(* Logix 5000 project; controller full_alarm_and_fault_management_system vendor 1 type 14 code 196 rev 36.11; software revision 36.00 *)

TASK MainTask (continuous, watchdog 500 ms) : MainProgram

MODULES
   Local : vendor 1 type 14 code 196 (5069 0, rev 36.11)
END_MODULES

PROGRAM MainProgram   (* main routine MainRoutine *)
VAR
   Active_Temp_SP : DINT;
   Code_EStop : DINT;   // 1001
   Code_HighLevel : DINT;   // 1005
   Code_HighTemp : DINT;   // 1003
   Code_LowLevel : DINT;   // 1006
   Code_LowTemp : DINT;   // 1004
   Code_MotorOL : DINT;   // 1002
   Code_SensorFault : DINT;   // 1010
   Code_Valve1Fail : DINT;   // 1007
   Code_Valve2Fail : DINT;   // 1008
   Code_Valve3Fail : DINT;   // 1009
   Current_Fault_Code : DINT;   // Optional displayed fault code
   Fault_Count : DINT;   // Optional number of active faults
   Flow_1_ok : BOOL;
   Flow_2_Ok : BOOL;
   Flow_3_ok : BOOL;
   Heat_Enable : BOOL;
   machine_Runpermissive : BOOL;
   ONS_EStop_TS : BOOL;   // One-shot storage for E-stop tiimestamping
   ONS_HighLevel_TS : BOOL;   // One-shot storage for high level timestamp
   ONS_HighTemp_TS : BOOL;   // One-shot storage for High temp timestamp
   ONS_LowLevel_TS : BOOL;   // One-shot storage for low level timestamp
   ONS_LowTemp_TS : BOOL;   // One-shot storage for low temp timestamp
   ONS_MotorOL_TS : BOOL;   // One-shot storage for motor overload timestamp
   ONS_Reset : BOOL;   // One-shot storage for reset pushbutton
   ONS_Sensor_TS : BOOL;   // One-shot storage for sensor fault timestamp
   ONS_Valve1_TS : BOOL;   // One-shot storage for valve 1 fault timestamp
   ONS_Valve2_TS : BOOL;   // One-shot storage for valve 2 fault timestamp
   ONS_Valve3_TS : BOOL;   // One-shot storage for valve 3 fault timestamp
   Sim_EStop_PB : BOOL;
   Sim_MotorOL : BOOL;
   system_run : BOOL;
   T_HeatTimeout : TIMER;
   Temp_PV : DINT;
   valve_1 : BOOL;
   valve_2 : BOOL;
   valve_3 : BOOL;
END_VAR
VAR_OUTPUT
   AlarmHorn : BOOL;   // Alarm output
   Any_Fault_Active : BOOL;   // True if any fault is latched
   Fault_Reset_Request : BOOL;   // One-shot reset request
   Flt_EStop : BOOL;   // Latched E-stop fault
   Flt_HighLevel : BOOL;   // Latched high level fault
   Flt_HighTemp : BOOL;   // Latched high temp fault
   Flt_LowLevel : BOOL;   // Latched low level fault
   Flt_LowTemp : BOOL;   // Latched low temp fault
   Flt_MotorOL : BOOL;   // Latched motor overload fault
   Flt_SensorFault : BOOL;   // Latched sensor fault
   Flt_Valve1Fail : BOOL;   // Latched valve 1 failure
   Flt_Valve2Fail : BOOL;   // latched valve 2 failure
   Flt_Valve3Fail : BOOL;   // Latched valve 3 failure
   Rst_OKLowLevel : BOOL;   // Low level cleared
   RstOk_EStop : BOOL;   // E-stop cleared, reset allowed
   RstOK_HighLevel : BOOL;   // High level cleared
   RstOK_HighTemp : BOOL;   // High temp cleared
   RstOK_LowTemp : BOOL;   // Low Temp cleared
   RstOk_motorOL : BOOL;   // Motor overload cleared
   RstOK_SensorFault : BOOL;   // sensor fault cleared
   RstOK_Valve1Fail : BOOL;   // Valve 1 fault cleared
   RstOK_Valve2Fail : BOOL;   // Valve 2 fault cleared
   RstOK_Valve3Fail : BOOL;   // Valve 3 fault cleared
   RTC_DateTime : DINT[7];   // Current controller time component
   TS_EStop : DINT[7];   // Timestamp for e-stop fault
   TS_HighLevel : DINT[7];   // Timestamp for high level
   TS_HighTemp : DINT[7];   // Timestamp for high temp
   TS_LowLevel : DINT[7];   // Timestamp for low level
   TS_LowTemp : DINT[7];   // Timestamp for low temp
   TS_MotorOL : DINT[7];   // Timestamp for motor overload
   TS_SensorFault : DINT[7];   // Timestamp for sensor fault
   TS_Valve1Fail : DINT[7];   // Timestamp for valve 1 fault
   TS_Valve2Fail : DINT[7];   // Timestamp for valve 2 Fault
   TS_Valve3Fail : DINT[7];   // Timestamp for valve 3 fault
END_VAR
VAR_INPUT
   Cond_EStop : BOOL;   // Raw E-stop condition
   Cond_Highlevel : BOOL;   // Raw high level fault
   Cond_HighTemp : BOOL;   // Raw high temperature fault
   Cond_Lowlevel : BOOL;   // Raw low level fault
   Cond_LowTemp : BOOL;   // Raw low temp fault
   Cond_MotorOL : BOOL;   // Raw motor overload condition
   Cond_SensorFault : BOOL;   // Raw valve 3 failure
   Cond_Valve1Fail : BOOL;   // Raw low level fault
   Cond_Valve2Fail : BOOL;   // Raw valve 1 failure
   Cond_Valve3Fail : BOOL;   // Raw valve 2 failure
   PB_AckFaults : BOOL;   // Optional acknowledge pushbutton
   PB_ResetFaults : BOOL;   // operator fault reset pushbutton
   Tank_level : DINT;
END_VAR

ROUTINE Fault_Detection   (* ladder *)
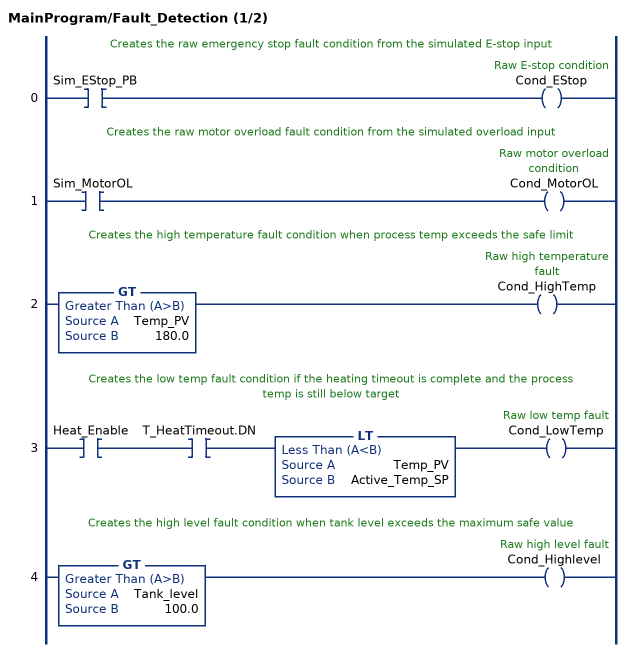
   // Creates the raw emergency stop fault condition from the simulated E-stop input
   0: XIC(Sim_EStop_PB)OTE(Cond_EStop);
   // Creates the raw motor overload fault condition from the simulated overload input
   1: XIC(Sim_MotorOL)OTE(Cond_MotorOL);
   // Creates the high temperature fault condition when process temp exceeds the safe limit
   2: GT(Temp_PV,180.0)OTE(Cond_HighTemp);
   // Creates the low temp fault condition if the heating timeout is complete and the process temp is still below target
   3: XIC(Heat_Enable)XIC(T_HeatTimeout.DN)LT(Temp_PV,Active_Temp_SP)OTE(Cond_LowTemp);
   // Creates the high level fault condition when tank level exceeds the maximum safe value
   4: GT(Tank_level,100.0)OTE(Cond_Highlevel);
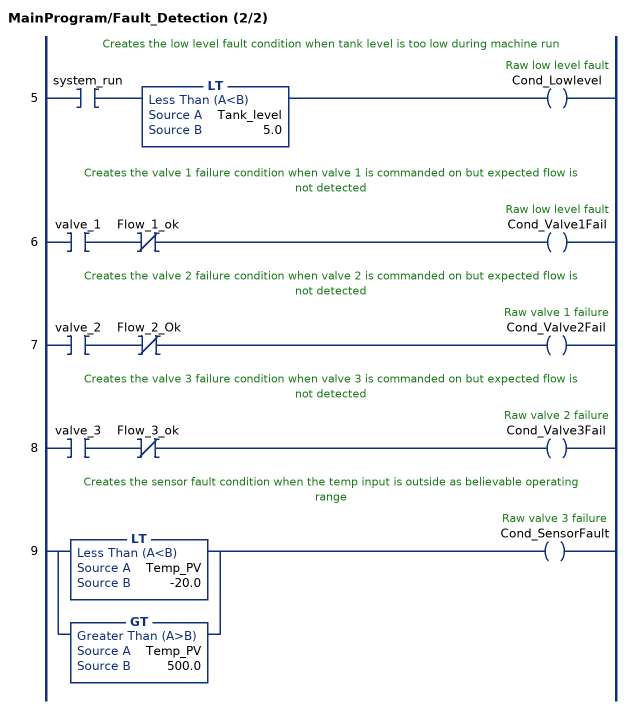
   // Creates the low level fault condition when tank level is too low during machine run
   5: XIC(system_run)LT(Tank_level,5.0)OTE(Cond_Lowlevel);
   // Creates the valve 1 failure condition when valve 1 is commanded on but expected flow is not detected
   6: XIC(valve_1)XIO(Flow_1_ok)OTE(Cond_Valve1Fail);
   // Creates the valve 2 failure condition when valve 2 is commanded on but expected flow is not detected
   7: XIC(valve_2)XIO(Flow_2_Ok)OTE(Cond_Valve2Fail);
   // Creates the valve 3 failure condition when valve 3 is commanded on but expected flow is not detected
   8: XIC(valve_3)XIO(Flow_3_ok)OTE(Cond_Valve3Fail);
   // Creates the sensor fault condition when the temp input is outside as believable operating range
   9: [LT(Temp_PV,-20.0) ,GT(Temp_PV,500.0) ]OTE(Cond_SensorFault);
END_ROUTINE

ROUTINE Fault_Display   (* ladder *)
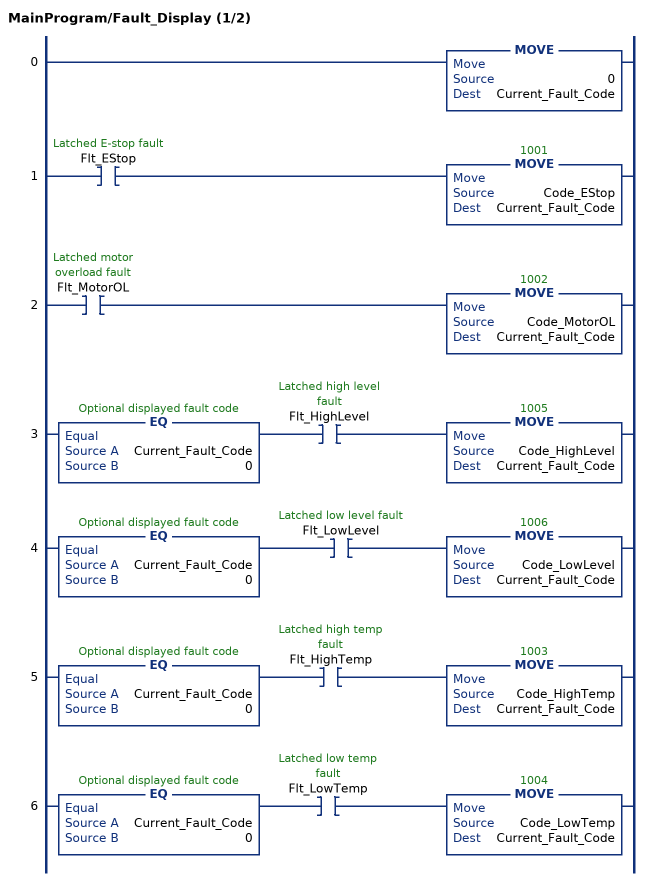
   0: MOVE(0,Current_Fault_Code);
   1: XIC(Flt_EStop)MOVE(Code_EStop,Current_Fault_Code);
   2: XIC(Flt_MotorOL)MOVE(Code_MotorOL,Current_Fault_Code);
   3: EQ(Current_Fault_Code,0)XIC(Flt_HighLevel)MOVE(Code_HighLevel,Current_Fault_Code);
   4: EQ(Current_Fault_Code,0)XIC(Flt_LowLevel)MOVE(Code_LowLevel,Current_Fault_Code);
   5: EQ(Current_Fault_Code,0)XIC(Flt_HighTemp)MOVE(Code_HighTemp,Current_Fault_Code);
   6: EQ(Current_Fault_Code,0)XIC(Flt_LowTemp)MOVE(Code_LowTemp,Current_Fault_Code);
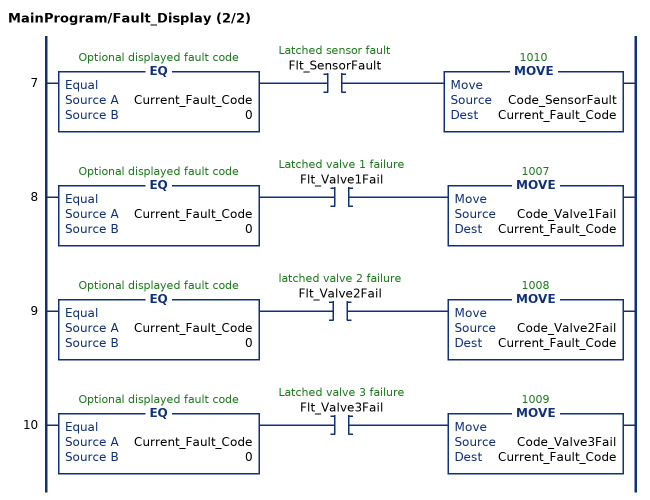
   7: EQ(Current_Fault_Code,0)XIC(Flt_SensorFault)MOVE(Code_SensorFault,Current_Fault_Code);
   8: EQ(Current_Fault_Code,0)XIC(Flt_Valve1Fail)MOVE(Code_Valve1Fail,Current_Fault_Code);
   9: EQ(Current_Fault_Code,0)XIC(Flt_Valve2Fail)MOVE(Code_Valve2Fail,Current_Fault_Code);
   10: EQ(Current_Fault_Code,0)XIC(Flt_Valve3Fail)MOVE(Code_Valve3Fail,Current_Fault_Code);
END_ROUTINE

ROUTINE Fault_Latching   (* ladder *)
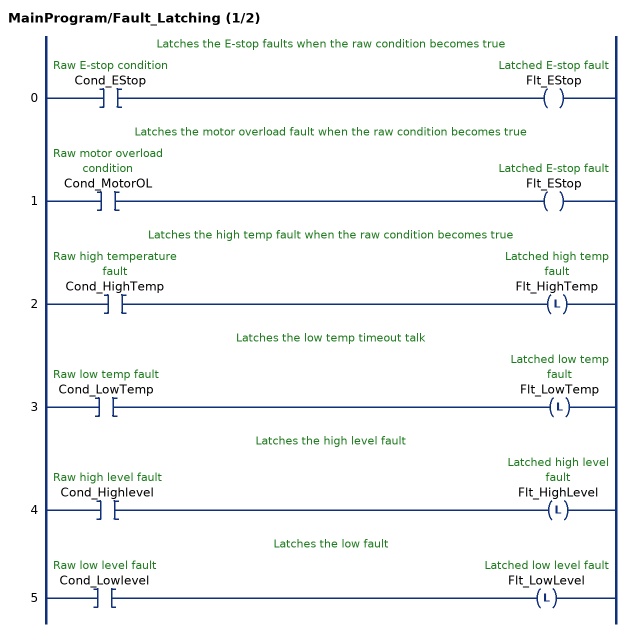
   // Latches the E-stop faults when the raw condition becomes true
   0: XIC(Cond_EStop)OTE(Flt_EStop);
   // Latches the motor overload fault when the raw condition becomes true
   1: XIC(Cond_MotorOL)OTE(Flt_EStop);
   // Latches the high temp fault when the raw condition becomes true
   2: XIC(Cond_HighTemp)OTL(Flt_HighTemp);
   // Latches the low temp timeout talk
   3: XIC(Cond_LowTemp)OTL(Flt_LowTemp);
   // Latches the high level fault
   4: XIC(Cond_Highlevel)OTL(Flt_HighLevel);
   // Latches the low fault
   5: XIC(Cond_Lowlevel)OTL(Flt_LowLevel);
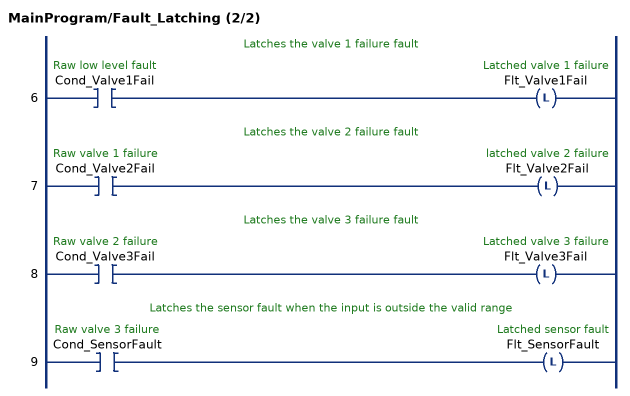
   // Latches the valve 1 failure fault
   6: XIC(Cond_Valve1Fail)OTL(Flt_Valve1Fail);
   // Latches the valve 2 failure fault
   7: XIC(Cond_Valve2Fail)OTL(Flt_Valve2Fail);
   // Latches the valve 3 failure fault
   8: XIC(Cond_Valve3Fail)OTL(Flt_Valve3Fail);
   // Latches the sensor fault when the input is outside the valid range
   9: XIC(Cond_SensorFault)OTL(Flt_SensorFault);
END_ROUTINE

ROUTINE Fault_Reset   (* ladder *)
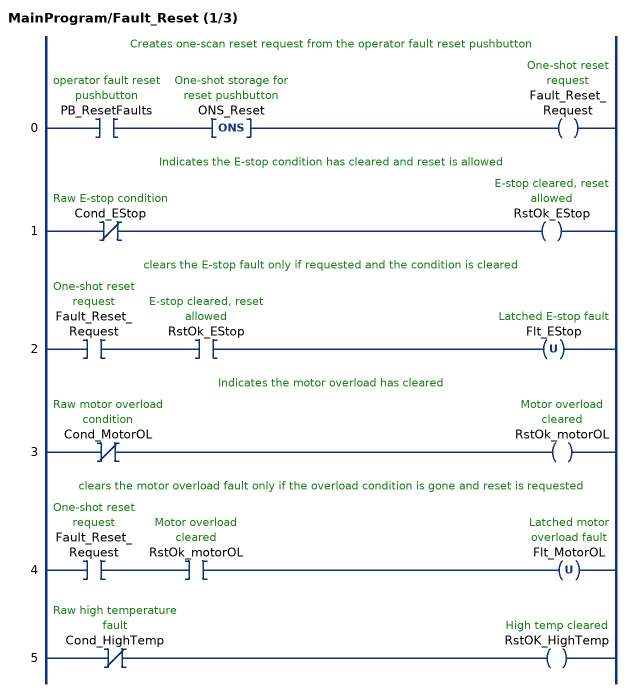
   // Creates one-scan reset request from the operator fault reset pushbutton
   0: XIC(PB_ResetFaults)ONS(ONS_Reset)OTE(Fault_Reset_Request);
   // Indicates the E-stop condition has cleared and reset is allowed
   1: XIO(Cond_EStop)OTE(RstOk_EStop);
   // clears the E-stop fault only if requested and the condition is cleared
   2: XIC(Fault_Reset_Request)XIC(RstOk_EStop)OTU(Flt_EStop);
   // Indicates the motor overload has cleared
   3: XIO(Cond_MotorOL)OTE(RstOk_motorOL);
   // clears the motor overload fault only if the overload condition is gone and reset is requested
   4: XIC(Fault_Reset_Request)XIC(RstOk_motorOL)OTU(Flt_MotorOL);
   5: XIO(Cond_HighTemp)OTE(RstOK_HighTemp);
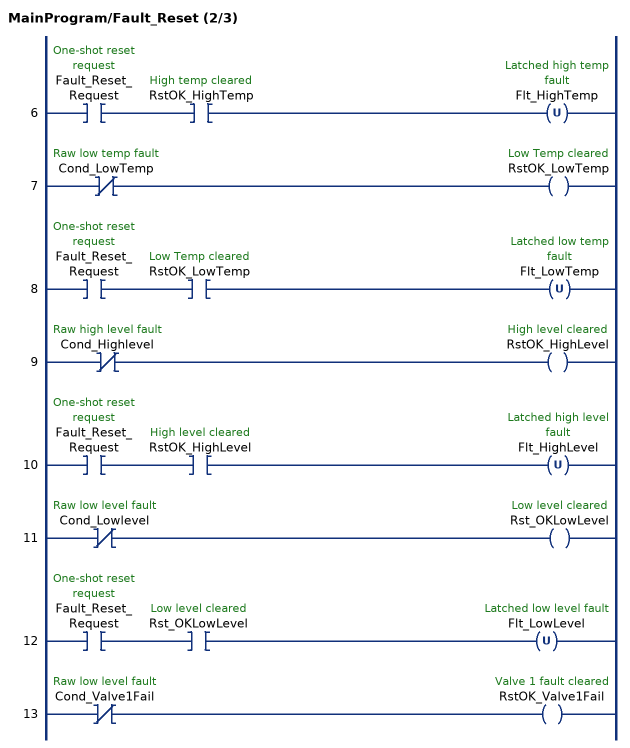
   6: XIC(Fault_Reset_Request)XIC(RstOK_HighTemp)OTU(Flt_HighTemp);
   7: XIO(Cond_LowTemp)OTE(RstOK_LowTemp);
   8: XIC(Fault_Reset_Request)XIC(RstOK_LowTemp)OTU(Flt_LowTemp);
   9: XIO(Cond_Highlevel)OTE(RstOK_HighLevel);
   10: XIC(Fault_Reset_Request)XIC(RstOK_HighLevel)OTU(Flt_HighLevel);
   11: XIO(Cond_Lowlevel)OTE(Rst_OKLowLevel);
   12: XIC(Fault_Reset_Request)XIC(Rst_OKLowLevel)OTU(Flt_LowLevel);
   13: XIO(Cond_Valve1Fail)OTE(RstOK_Valve1Fail);
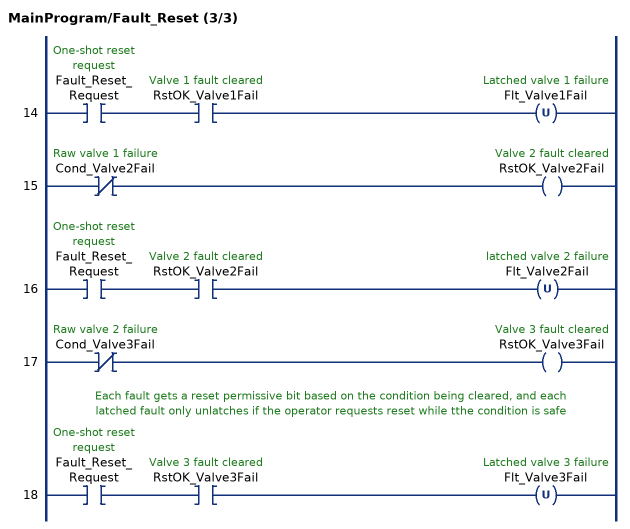
   14: XIC(Fault_Reset_Request)XIC(RstOK_Valve1Fail)OTU(Flt_Valve1Fail);
   15: XIO(Cond_Valve2Fail)OTE(RstOK_Valve2Fail);
   16: XIC(Fault_Reset_Request)XIC(RstOK_Valve2Fail)OTU(Flt_Valve2Fail);
   17: XIO(Cond_Valve3Fail)OTE(RstOK_Valve3Fail);
   // Each fault gets a reset permissive bit based on the condition being cleared, and each latched fault only unlatches if the operator requests reset while tthe condition is safe
   18: XIC(Fault_Reset_Request)XIC(RstOK_Valve3Fail)OTU(Flt_Valve3Fail);
END_ROUTINE

ROUTINE Fault_summary   (* ladder *)
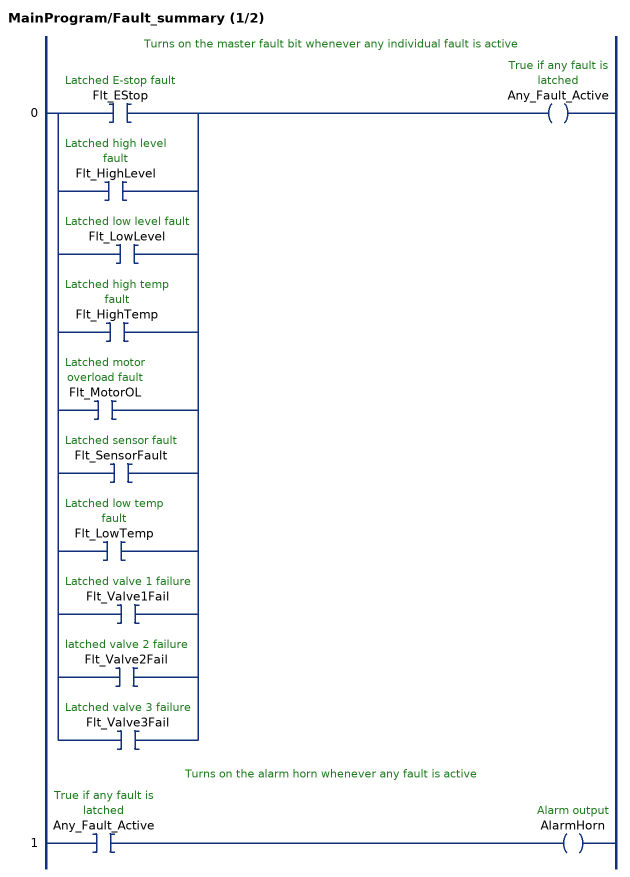
   // Turns on the master fault bit whenever any individual fault is active
   0: [XIC(Flt_EStop) ,XIC(Flt_HighLevel) ,XIC(Flt_LowLevel) ,XIC(Flt_HighTemp) ,XIC(Flt_MotorOL) ,XIC(Flt_SensorFault) ,XIC(Flt_LowTemp) ,XIC(Flt_Valve1Fail) ,XIC(Flt_Valve2Fail) ,XIC(Flt_Valve3Fail) ]OTE(Any_Fault_Active);
   // Turns on the alarm horn whenever any fault is active
   1: XIC(Any_Fault_Active)OTE(AlarmHorn);
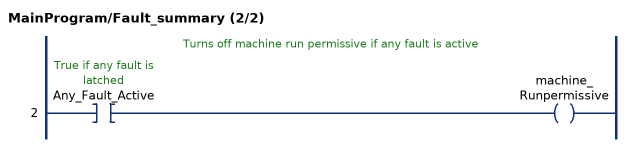
   // Turns off machine run permissive if any fault is active
   2: XIC(Any_Fault_Active)OTE(machine_Runpermissive);
END_ROUTINE

ROUTINE Fault_Timestamps   (* ladder *)
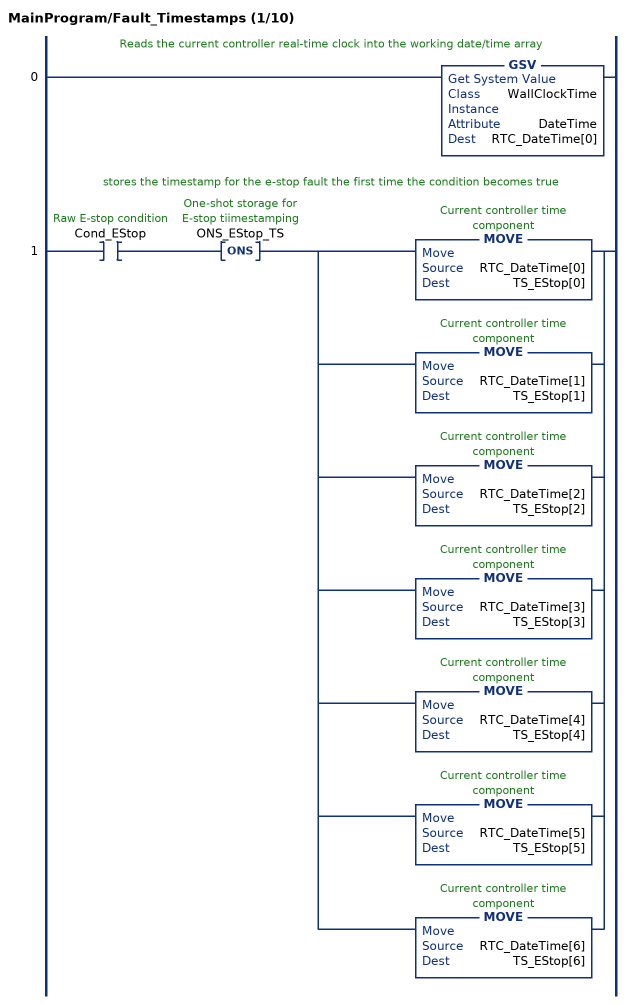
   // Reads the current controller real-time clock into the working date/time array
   0: GSV(WallClockTime,,DateTime,RTC_DateTime[0]);
   // stores the timestamp for the e-stop fault the first time the condition becomes true
   1: XIC(Cond_EStop)ONS(ONS_EStop_TS)[MOVE(RTC_DateTime[0],TS_EStop[0]) ,MOVE(RTC_DateTime[1],TS_EStop[1]) ,MOVE(RTC_DateTime[2],TS_EStop[2]) ,MOVE(RTC_DateTime[3],TS_EStop[3]) ,MOVE(RTC_DateTime[4],TS_EStop[4]) ,MOVE(RTC_DateTime[5],TS_EStop[5]) ,MOVE(RTC_DateTime[6],TS_EStop[6]) ];
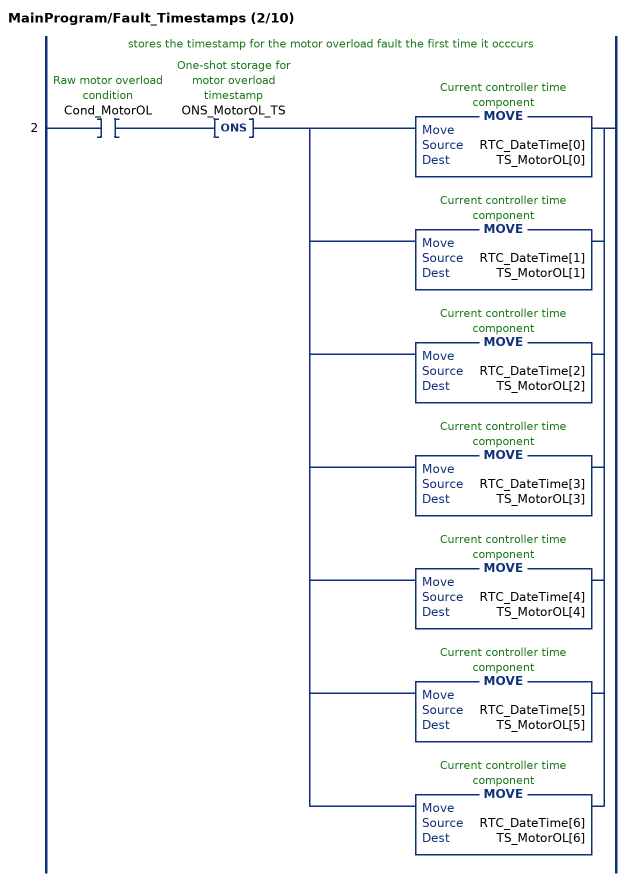
   // stores the timestamp for the motor overload fault the first time it occcurs
   2: XIC(Cond_MotorOL)ONS(ONS_MotorOL_TS)[MOVE(RTC_DateTime[0],TS_MotorOL[0]) ,MOVE(RTC_DateTime[1],TS_MotorOL[1]) ,MOVE(RTC_DateTime[2],TS_MotorOL[2]) ,MOVE(RTC_DateTime[3],TS_MotorOL[3]) ,MOVE(RTC_DateTime[4],TS_MotorOL[4]) ,MOVE(RTC_DateTime[5],TS_MotorOL[5]) ,MOVE(RTC_DateTime[6],TS_MotorOL[6]) ];
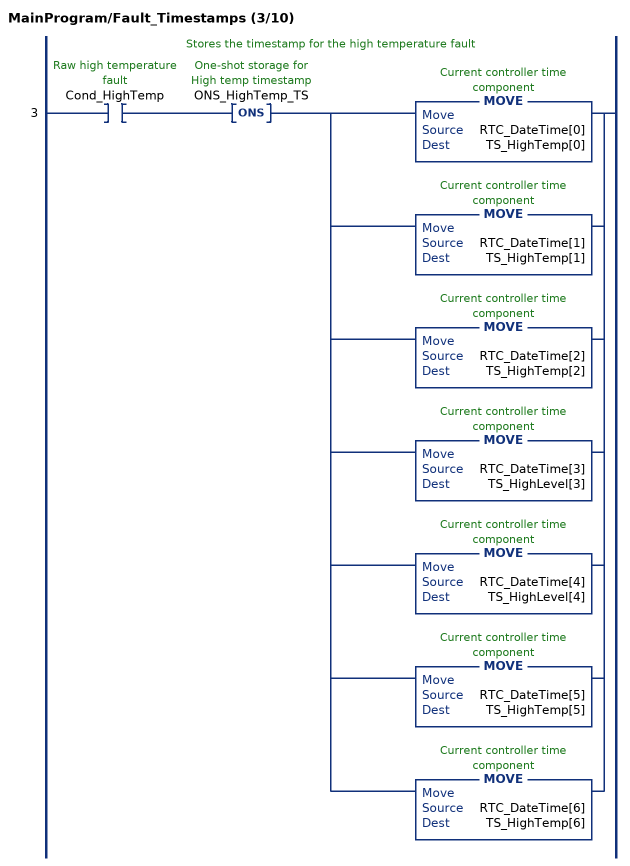
   // Stores the timestamp for the high temperature fault
   3: XIC(Cond_HighTemp)ONS(ONS_HighTemp_TS)[MOVE(RTC_DateTime[0],TS_HighTemp[0]) ,MOVE(RTC_DateTime[1],TS_HighTemp[1]) ,MOVE(RTC_DateTime[2],TS_HighTemp[2]) ,MOVE(RTC_DateTime[3],TS_HighLevel[3]) ,MOVE(RTC_DateTime[4],TS_HighLevel[4]) ,MOVE(RTC_DateTime[5],TS_HighTemp[5]) ,MOVE(RTC_DateTime[6],TS_HighTemp[6]) ];
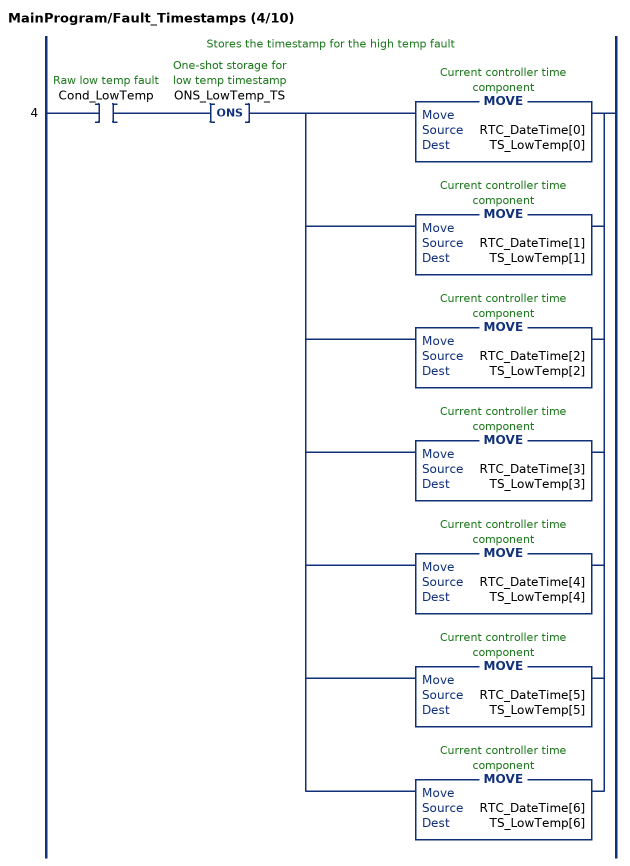
   // Stores the timestamp for the high temp fault
   4: XIC(Cond_LowTemp)ONS(ONS_LowTemp_TS)[MOVE(RTC_DateTime[0],TS_LowTemp[0]) ,MOVE(RTC_DateTime[1],TS_LowTemp[1]) ,MOVE(RTC_DateTime[2],TS_LowTemp[2]) ,MOVE(RTC_DateTime[3],TS_LowTemp[3]) ,MOVE(RTC_DateTime[4],TS_LowTemp[4]) ,MOVE(RTC_DateTime[5],TS_LowTemp[5]) ,MOVE(RTC_DateTime[6],TS_LowTemp[6]) ];
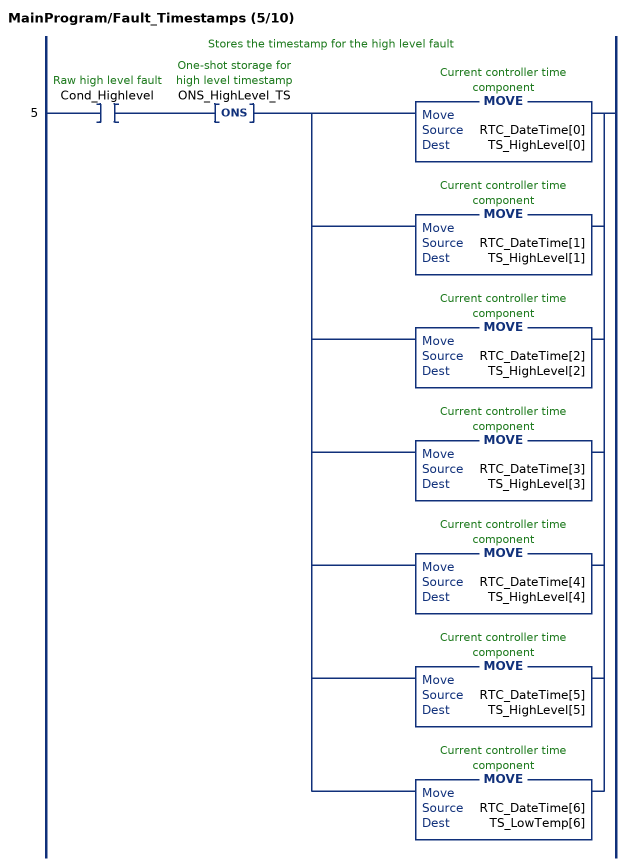
   // Stores the timestamp for the high level fault
   5: XIC(Cond_Highlevel)ONS(ONS_HighLevel_TS)[MOVE(RTC_DateTime[0],TS_HighLevel[0]) ,MOVE(RTC_DateTime[1],TS_HighLevel[1]) ,MOVE(RTC_DateTime[2],TS_HighLevel[2]) ,MOVE(RTC_DateTime[3],TS_HighLevel[3]) ,MOVE(RTC_DateTime[4],TS_HighLevel[4]) ,MOVE(RTC_DateTime[5],TS_HighLevel[5]) ,MOVE(RTC_DateTime[6],TS_LowTemp[6]) ];
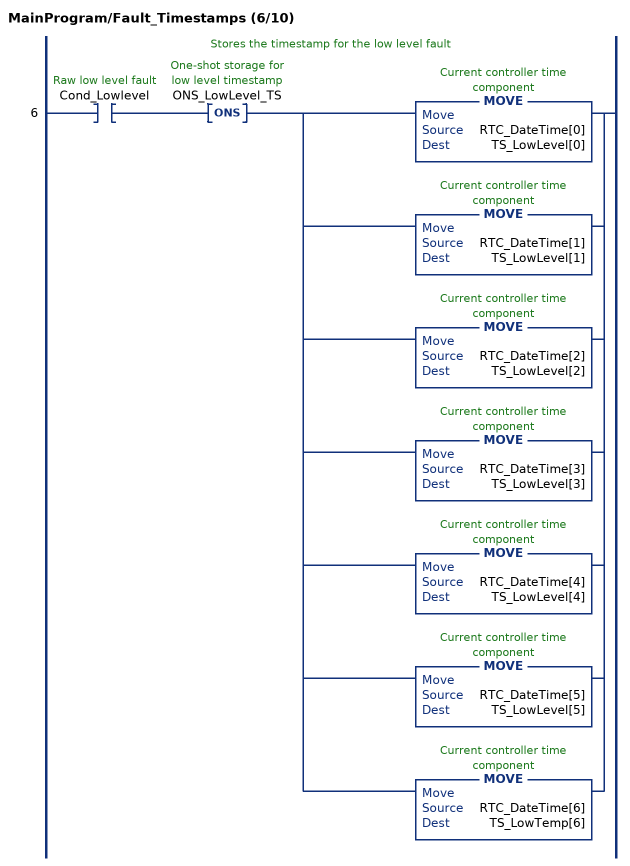
   // Stores the timestamp for the low level fault
   6: XIC(Cond_Lowlevel)ONS(ONS_LowLevel_TS)[MOVE(RTC_DateTime[0],TS_LowLevel[0]) ,MOVE(RTC_DateTime[1],TS_LowLevel[1]) ,MOVE(RTC_DateTime[2],TS_LowLevel[2]) ,MOVE(RTC_DateTime[3],TS_LowLevel[3]) ,MOVE(RTC_DateTime[4],TS_LowLevel[4]) ,MOVE(RTC_DateTime[5],TS_LowLevel[5]) ,MOVE(RTC_DateTime[6],TS_LowTemp[6]) ];
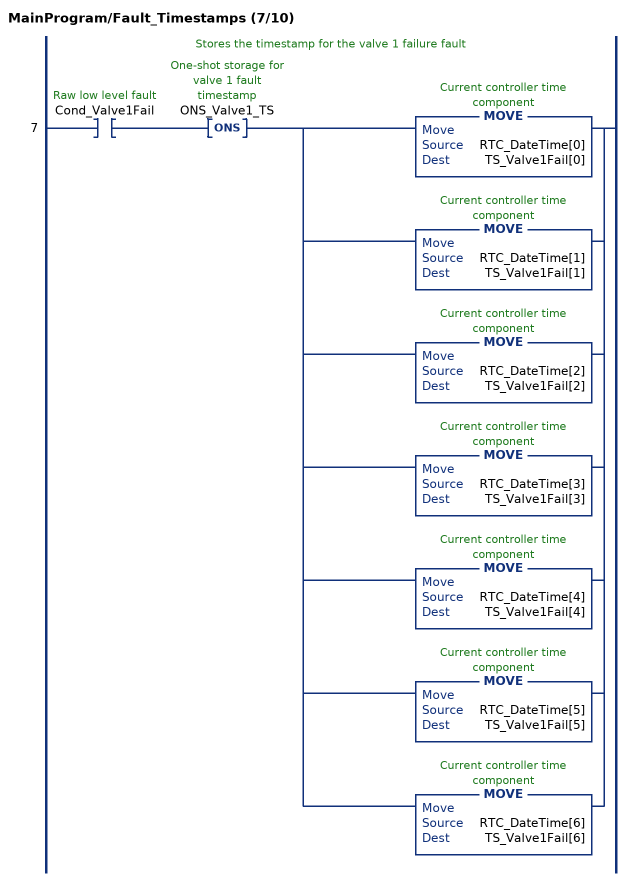
   // Stores the timestamp for the valve 1 failure fault
   7: XIC(Cond_Valve1Fail)ONS(ONS_Valve1_TS)[MOVE(RTC_DateTime[0],TS_Valve1Fail[0]) ,MOVE(RTC_DateTime[1],TS_Valve1Fail[1]) ,MOVE(RTC_DateTime[2],TS_Valve1Fail[2]) ,MOVE(RTC_DateTime[3],TS_Valve1Fail[3]) ,MOVE(RTC_DateTime[4],TS_Valve1Fail[4]) ,MOVE(RTC_DateTime[5],TS_Valve1Fail[5]) ,MOVE(RTC_DateTime[6],TS_Valve1Fail[6]) ];
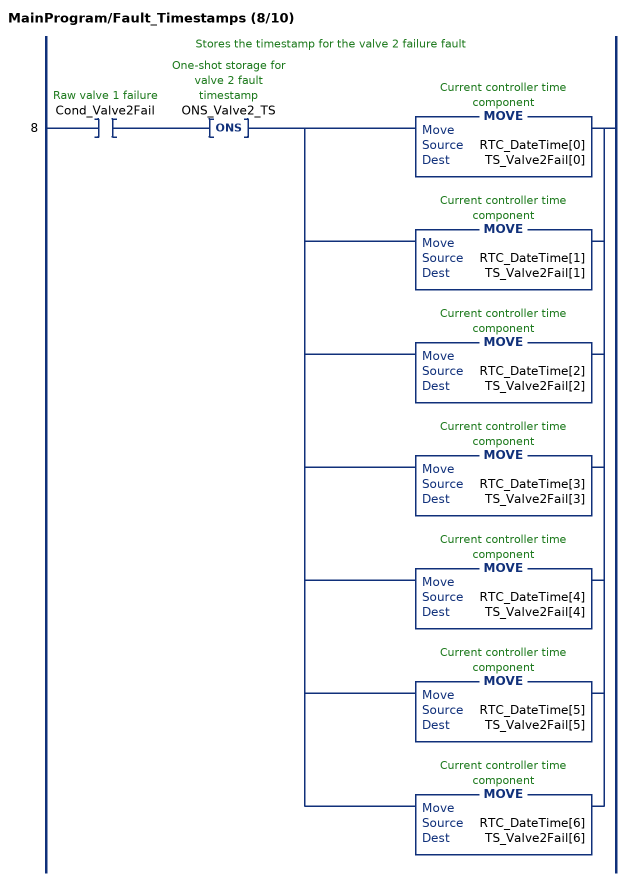
   // Stores the timestamp for the valve 2 failure fault
   8: XIC(Cond_Valve2Fail)ONS(ONS_Valve2_TS)[MOVE(RTC_DateTime[0],TS_Valve2Fail[0]) ,MOVE(RTC_DateTime[1],TS_Valve2Fail[1]) ,MOVE(RTC_DateTime[2],TS_Valve2Fail[2]) ,MOVE(RTC_DateTime[3],TS_Valve2Fail[3]) ,MOVE(RTC_DateTime[4],TS_Valve2Fail[4]) ,MOVE(RTC_DateTime[5],TS_Valve2Fail[5]) ,MOVE(RTC_DateTime[6],TS_Valve2Fail[6]) ];
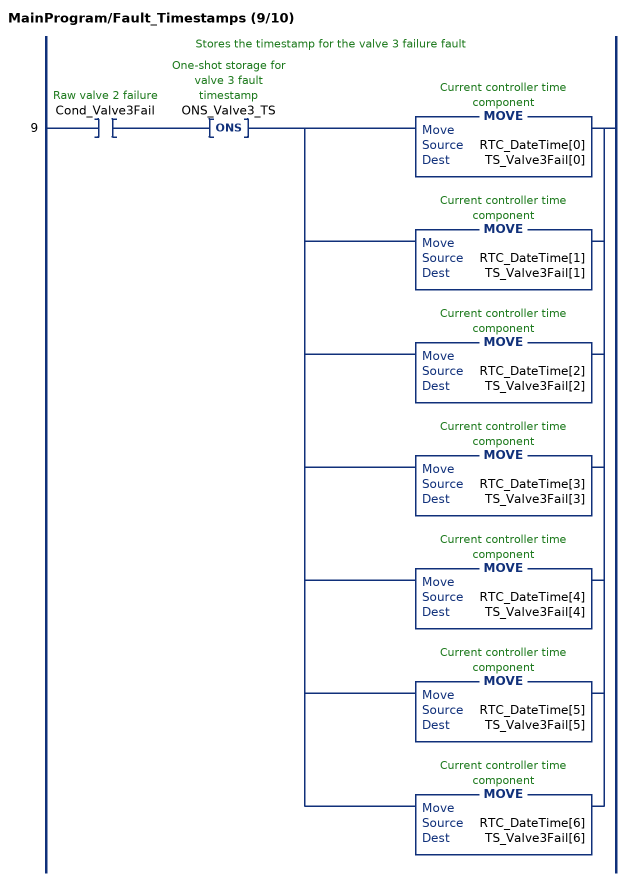
   // Stores the timestamp for the valve 3 failure fault
   9: XIC(Cond_Valve3Fail)ONS(ONS_Valve3_TS)[MOVE(RTC_DateTime[0],TS_Valve3Fail[0]) ,MOVE(RTC_DateTime[1],TS_Valve3Fail[1]) ,MOVE(RTC_DateTime[2],TS_Valve3Fail[2]) ,MOVE(RTC_DateTime[3],TS_Valve3Fail[3]) ,MOVE(RTC_DateTime[4],TS_Valve3Fail[4]) ,MOVE(RTC_DateTime[5],TS_Valve3Fail[5]) ,MOVE(RTC_DateTime[6],TS_Valve3Fail[6]) ];
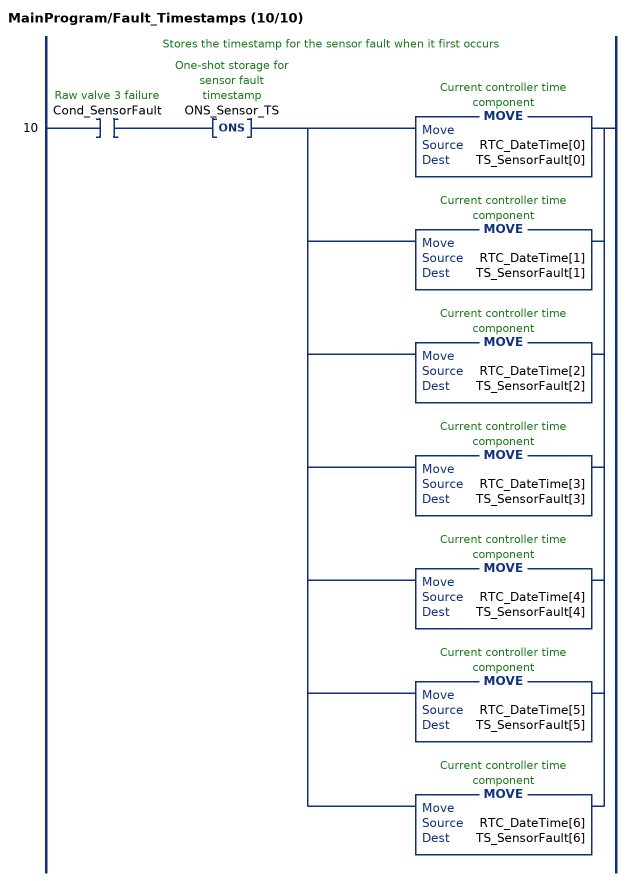
   // Stores the timestamp for the sensor fault when it first occurs
   10: XIC(Cond_SensorFault)ONS(ONS_Sensor_TS)[MOVE(RTC_DateTime[0],TS_SensorFault[0]) ,MOVE(RTC_DateTime[1],TS_SensorFault[1]) ,MOVE(RTC_DateTime[2],TS_SensorFault[2]) ,MOVE(RTC_DateTime[3],TS_SensorFault[3]) ,MOVE(RTC_DateTime[4],TS_SensorFault[4]) ,MOVE(RTC_DateTime[5],TS_SensorFault[5]) ,MOVE(RTC_DateTime[6],TS_SensorFault[6]) ];
END_ROUTINE

ROUTINE MainRoutine   (* ladder *)
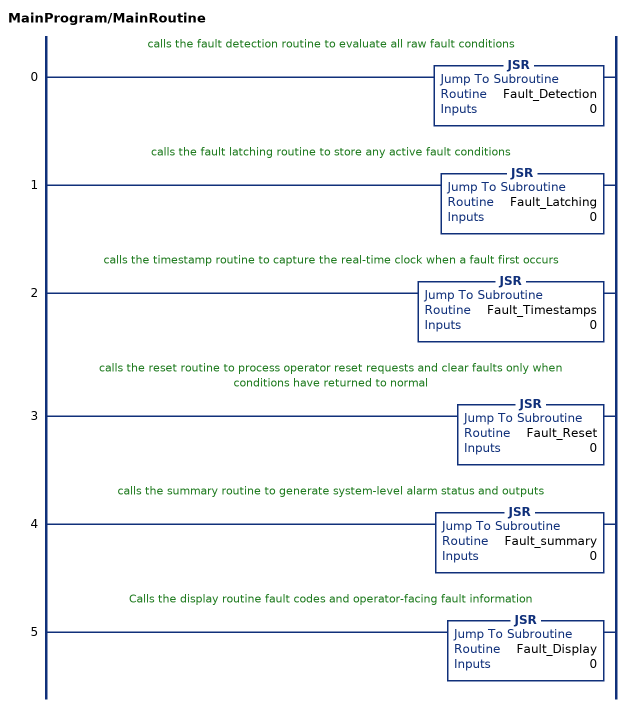
   // calls the fault detection routine to evaluate all raw fault conditions
   0: JSR(Fault_Detection,0);
   // calls the fault latching routine to store any active fault conditions
   1: JSR(Fault_Latching,0);
   // calls the timestamp routine to capture the real-time clock when a fault first occurs
   2: JSR(Fault_Timestamps,0);
   // calls the reset routine to process operator reset requests and clear faults only when conditions have returned to normal
   3: JSR(Fault_Reset,0);
   // calls the summary routine to generate system-level alarm status and outputs
   4: JSR(Fault_summary,0);
   // Calls the display routine fault codes and operator-facing fault information
   5: JSR(Fault_Display,0);
END_ROUTINE
END_PROGRAM
